{attribute 'qualified_only'}
{attribute 'strict'}
TYPE EFeedbackMsgPhotoLumChamber :
(
	InterlockPanelsMsg := 20,
	SlitDoorPositionMsg := 30,
	SlitDoorOpenPositionMsg,
	SlitDoorClosePositionMsg
);
END_TYPE

(* stored: Version 1.1.0.1, ProductVersion 3.1.4024.12
   DUT EFeedbackMsgPhotoLumChamber: Id {e916dbf7-d904-462d-8bb0-9d84796f2191} *)
